// TIA Portal project "SELECTOR" (V16)

(* hardware
DEVICE "S7-1200 station_1"  S7-1200 Station
   slot 0: "Rack_0"  S7-1200 Rack  Rack  V1.0
   slot 1: "PLC_1"  CPU 1212C AC/DC/Rly  6ES7 212-1BE40-0XB0  V4.4
*)

// ===== PLC "PLC_1"  CPU 1212C AC/DC/Rly =====

VAR_GLOBAL   // PLC tag table "Default tag table"
   "START" AT %I0.0 : Bool;
   "STOP" AT %I0.1 : Bool;
   "MOTOR1" AT %Q0.0 : Bool;
   "MOTOR2" AT %Q0.1 : Bool;
   "MOTOR3" AT %Q0.2 : Bool;
   "SELECT A" AT %I0.2 : Bool;
   "SELECT B" AT %I0.3 : Bool;
   "X" AT %M0.0 : Bool;
   "NO SEKECT" AT %M0.1 : Bool;
   "TM1" AT %M0.2 : Bool;
   "TM2" AT %M0.3 : Bool;
END_VAR

// folder: System blocks/Program resources

DATA_BLOCK "T1"   // DB1
{ S7_Optimized_Access := 'TRUE' }
AUTHOR : Simatic
FAMILY : IEC
NAME : IEC_TMR
VERSION : 1.0
// stored: InstanceOfName IEC_TIMER
"IEC_TIMER"
BEGIN
END_DATA_BLOCK

DATA_BLOCK "T2"   // DB2
{ S7_Optimized_Access := 'TRUE' }
AUTHOR : Simatic
FAMILY : IEC
NAME : IEC_TMR
VERSION : 1.0
// stored: InstanceOfName IEC_TIMER
"IEC_TIMER"
BEGIN
END_DATA_BLOCK

// folder: (top level)

ORGANIZATION_BLOCK "Main"   // OB1, LAD, ProgramCycle
TITLE = "Main Program Sweep (Cycle)"
{ S7_Optimized_Access := 'TRUE' }
VERSION : 0.1
   VAR_INPUT
      Initial_Call : Bool;   // Initial call of this OB
      Remanence : Bool;   // =True, if remanent data are available
   END_VAR
BEGIN

REGION Network 1
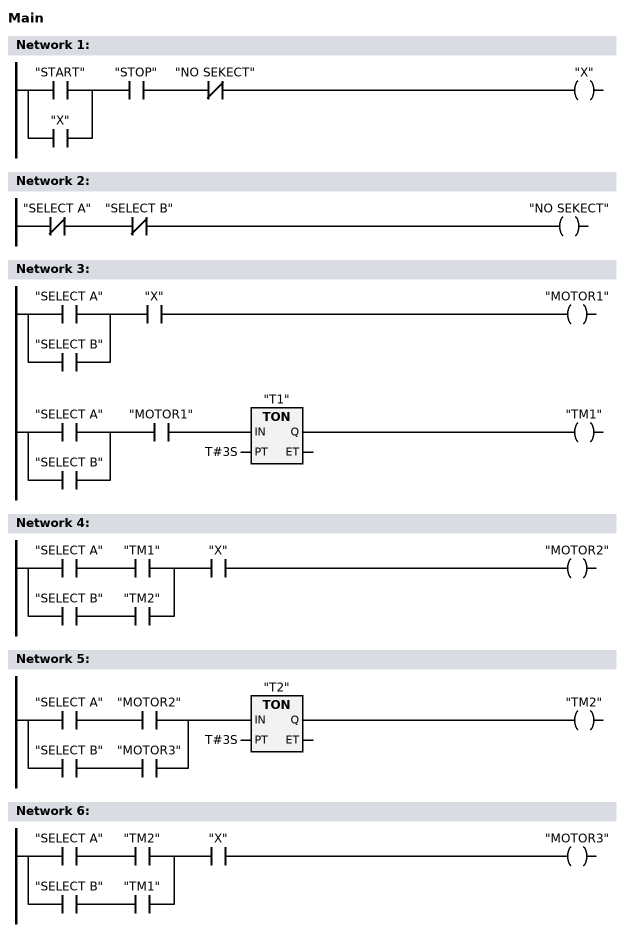
   RUNG wire#powerrail
      Contact( "START" )
      wire#w1
      Contact( "STOP" )
      I_Contact( "NO SEKECT" )
      Coil( "X" )
   END_RUNG
   RUNG wire#powerrail
      Contact( "X" )
   END_RUNG wire#w1
   // the same network as SCL:
   "X" := ("START" OR "X") AND "STOP" AND NOT "NO SEKECT";
END_REGION

REGION Network 2
   RUNG wire#powerrail
      I_Contact( "SELECT A" )
      I_Contact( "SELECT B" )
      Coil( "NO SEKECT" )
   END_RUNG
   // the same network as SCL:
   "NO SEKECT" := NOT "SELECT A" AND NOT "SELECT B";
END_REGION

REGION Network 3
   "MOTOR1" := ("SELECT A" OR "SELECT B") AND "X";
   "T1".TON(IN := ("SELECT A" OR "SELECT B") AND "MOTOR1", PT := T#3S);
   "TM1" := "T1".Q;
END_REGION

REGION Network 4
   RUNG wire#powerrail
      Contact( "SELECT A" )
      Contact( "TM1" )
      wire#w1
      Contact( "X" )
      Coil( "MOTOR2" )
   END_RUNG
   RUNG wire#powerrail
      Contact( "SELECT B" )
      Contact( "TM2" )
   END_RUNG wire#w1
   // the same network as SCL:
   "MOTOR2" := (("SELECT A" AND "TM1") OR ("SELECT B" AND "TM2")) AND "X";
END_REGION

REGION Network 5
   "T2".TON(IN := ("SELECT A" AND "MOTOR2") OR ("SELECT B" AND "MOTOR3"), PT := T#3S);
   "TM2" := "T2".Q;
END_REGION

REGION Network 6
   RUNG wire#powerrail
      Contact( "SELECT A" )
      Contact( "TM2" )
      wire#w1
      Contact( "X" )
      Coil( "MOTOR3" )
   END_RUNG
   RUNG wire#powerrail
      Contact( "SELECT B" )
      Contact( "TM1" )
   END_RUNG wire#w1
   // the same network as SCL:
   "MOTOR3" := (("SELECT A" AND "TM2") OR ("SELECT B" AND "TM1")) AND "X";
END_REGION
END_ORGANIZATION_BLOCK